# EPICS autosave request: 3-3/GalilSup/Db/galil_user_array.req
# User array settings
$(P)UARRAYNAME0_SP
$(P)UARRAYNAME1_SP
$(P)UARRAYNAME2_SP
$(P)UARRAYNAME3_SP
$(P)UARRAYNAME4_SP
$(P)UARRAYNAME5_SP
$(P)UARRAYNAME6_SP
$(P)UARRAYNAME7_SP
